{attribute addProperty BoxType "EP5001-0002-0016"}
{attribute addProperty Id "SSI_InputsAT %I*SSI_Inputs_C03DB35B4860WcStateAT %I*WcState_F855686C1620InfoDataAT %I*InfoData_BC63D37F80100"}
{attribute addProperty CRC "1624121117"}
{attribute addProperty SizeInBites "144"}
{attribute addProperty SizeInBytes "18"}
TYPE EP5001_636E7B50 :
STRUCT
	{attribute addProperty Name "SSI_Inputs"}
	SSI_Inputs : SSI_Inputs_C03DB35B;
	{attribute addProperty Name "WcState"}
	WcState : WcState_F855686C;
	{attribute addProperty Name "InfoData"}
	InfoData : InfoData_BC63D37F;
END_STRUCT
END_TYPE

(* stored: Version 1.2.0.0, ProductVersion 3.1.4024.9
   DUT EP5001_636E7B50: Id {a9db2b1a-1be5-478b-9d60-3d92a59ea6f1} *)
